Universal Robots PolyScope program: 1ac.urp

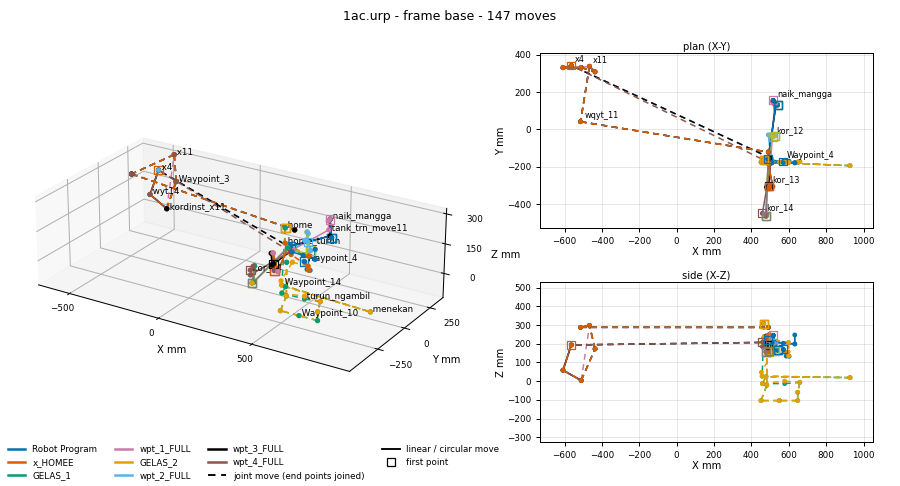
[picture p0: tool path of 1ac.urp in frame base, 147 of 147 moves have a stored position in this frame; points joined in program order, loops and branches not executed]
Program 1ac (createdIn=3.4.3.361 lastSavedIn=3.4.3.361 directory=/programs installation=default robotSerialNumber=2017332896)
Calibrated DH parameters: a=[0.000025, -0.243644, -0.213352, 0.00001, -0.000078, 0]; d=[0.152306, -2.943792, 4.680366, -1.624115, 0.085414, 0.082498]; alpha=[1.571129, 0.003245, -0.003887, 1.571551, -1.571075, 0]; deltaTheta=[0.000074, -0.039266, 0.00755, 0.031605, -0.000097, -0.000018]
BeforeStart
  komunikasi := socket_open("192.168.0.120",30002)
  count := 0
Robot Program (runOnlyOnce=false motionType=MoveJ speed=1.047198 acceleration=1.396263 useActiveTCP=false)
  MoveJ speed 60 deg/s, acceleration 80 deg/s^2 (useActiveTCP=false)
    SuppressedNode
      Waypoint x_HOME: TCP in base x=391.792 y=-168.42 z=273.232 mm, rx=2.1755 ry=-0.1538 rz=2.2323 rad; joints [-13.452, -76.313, -113.498, -168.909, -98.804, -86.905] deg; flange x=205.883 y=-152.538 z=268.8 mm, rx=0.1091 ry=1.5439 rz=-0.0229 rad
    URCap RG2 (RG2 - On Robot, On Robot ApS) data=depthCompensate = false
      | width = 0
      | name = RG2(0)
      | force = 40
      | trigIsDefined = 1
  Loop While (checkContinuously=false) expression=komunikasi≟ False
    komunikasi := socket_open("192.168.0.120",30002)
    If digital_in[7]≟ False
      MoveJ speed 60 deg/s, acceleration 80 deg/s^2 (useActiveTCP=false)
        Waypoint Waypoint_4: TCP in base x=570.948 y=-172.227 z=170.703 mm, rx=1.2117 ry=1.0902 rz=1.141 rad; joints [-5.248, -122.842, -90.085, -143.869, -88.947, -540.731] deg; flange x=385.83 y=-150.884 z=160.264 mm, rx=-1.1206 ry=1.2455 rz=-1.3283 rad
        Waypoint Waypoint_5: TCP in base x=571.886 y=-168.478 z=167.165 mm, rx=0.1353 ry=1.5152 rz=-0.0293 rad; joints [-4.915, -123.143, -90.137, -143.887, -89.039, -626.132] deg; flange x=386.547 y=-148.493 z=157.904 mm, rx=2.1391 ry=-0.191 rz=2.2564 rad
        Waypoint Waypoint_7: TCP in base x=585.683 y=-169.223 z=134.026 mm, rx=0.0805 ry=1.5489 rz=0.0242 rad; joints [-8.112, -130.965, -83.945, -143.962, -96.278, -626.137] deg; flange x=399.213 y=-162.362 z=130.346 mm, rx=-2.181 ry=0.1133 rz=-2.2277 rad
        Waypoint Waypoint_15: TCP in base x=601.355 y=-170.35 z=133.169 mm, rx=0.1182 ry=1.5455 rz=-0.0126 rad; joints [-5.838, -133.147, -80.115, -145.564, -91.253, -626.166] deg; flange x=415.411 y=-154.657 z=129.279 mm, rx=2.184 ry=-0.1672 rz=2.2361 rad
        Wait DigitalInput pin=digital_in[7]; digitalValue=0
    Wait Sleep waitTime=0.5
  pose_position := get_actual_tcp_pose()
  joint_positions := get_actual_joint_positions()
  Script: socket_send_string(pose_position)
  Wait Sleep waitTime=0.5
  Script: socket_send_string(joint_positions)
  Wait Sleep waitTime=0.5
  Script: socket_send_string("asking_for_data")
  Wait Sleep waitTime=0.5
  dt_kirim := socket_read_ascii_float(1)
  dt_terima := dt_kirim[1]
  Wait Sleep waitTime=0.5
  komunikasi := False
  Script: socket_close()
  Folder Folder
    '1'
    If komunikasi≟ False
      If dt_terima≟1
        MoveJ speed 60 deg/s, acceleration 80 deg/s^2 (useActiveTCP=false)
          If digital_in[4]≟ False
            Call GELAS_1
            Call wpt_1_FULL
          ElseIf digital_in[4]≟ True
            Call GELAS_2
            Call wpt_1_FULL
        dt_terima := 0
      If dt_terima≟2
        MoveJ speed 60 deg/s, acceleration 80 deg/s^2 (useActiveTCP=false)
          If digital_in[4]≟ False
            Call GELAS_1
            Call wpt_2_FULL
          ElseIf digital_in[4]≟ True
            Call GELAS_2
            Call wpt_2_FULL
          dt_terima := 0
      If dt_terima≟3
        MoveJ speed 60 deg/s, acceleration 80 deg/s^2 (useActiveTCP=false)
          If digital_in[4]≟ False
            Call GELAS_1
            Call wpt_3_FULL
          ElseIf digital_in[4]≟ True
            Call GELAS_2
            Call wpt_3_FULL
          dt_terima := 0
      If dt_terima≟4
        MoveJ speed 60 deg/s, acceleration 80 deg/s^2 (useActiveTCP=false)
          If digital_in[4]≟ False
            Call GELAS_1
            Call wpt_4_FULL
          ElseIf digital_in[4]≟ True
            Call GELAS_2
            Call wpt_4_FULL
          dt_terima := 0
      '50=50'
      If dt_terima≟5
        'mangga'
        MoveJ speed 60 deg/s, acceleration 80 deg/s^2 (useActiveTCP=false)
          If digital_in[4]≟ False
            Call GELAS_1
            Call manga50
            Call melon50
            Call mixer
            Call x_to_pelanggan
          ElseIf digital_in[4]≟ True
            Call GELAS_2
            Call manga50
            Call melon50
            Call mixer
            Call x_to_pelanggan
          dt_terima := 0
      If dt_terima≟6
        MoveJ speed 60 deg/s, acceleration 80 deg/s^2 (useActiveTCP=false)
          If digital_in[4]≟ False
            Call GELAS_1
            Call manga50
            Call melon50
            Call mixer
            Call x_to_pelanggan
          ElseIf digital_in[4]≟ True
            Call GELAS_2
            Call manga50
            Call melon50
            Call mixer
            Call x_to_pelanggan
          dt_terima := 0
      If dt_terima≟7
        MoveJ speed 60 deg/s, acceleration 80 deg/s^2 (useActiveTCP=false)
          If digital_in[4]≟ False
            Call GELAS_1
            Call manga50
            Call cc_pandan50
            Call mixer
            Call x_to_pelanggan
          ElseIf digital_in[4]≟ True
            Call GELAS_2
            Call manga50
            Call cc_pandan50
            Call mixer
            Call x_to_pelanggan
          dt_terima := 0
      If dt_terima≟8
        MoveJ speed 60 deg/s, acceleration 80 deg/s^2 (useActiveTCP=false)
          If digital_in[4]≟ False
            Call GELAS_1
            Call melon50
            Call jeruk50
            Call mixer
            Call x_to_pelanggan
          ElseIf digital_in[4]≟ True
            Call GELAS_2
            Call melon50
            Call jeruk50
            Call mixer
            Call x_to_pelanggan
          dt_terima := 0
      If dt_terima≟9
        MoveJ speed 60 deg/s, acceleration 80 deg/s^2 (useActiveTCP=false)
          If digital_in[4]≟ False
            Call GELAS_1
            Call melon50
            Call cc_pandan50
            Call mixer
            Call x_to_pelanggan
          ElseIf digital_in[4]≟ True
            Call GELAS_2
            Call melon50
            Call cc_pandan50
            Call mixer
            Call x_to_pelanggan
          count := 0
      If dt_terima≟10
        MoveJ speed 60 deg/s, acceleration 80 deg/s^2 (useActiveTCP=false)
          If digital_in[4]≟ False
            Call GELAS_1
            Call melon50
            Call manga50
            Call mixer
            Call x_to_pelanggan
          ElseIf digital_in[4]≟ True
            Call GELAS_2
            Call melon50
            Call manga50
            Call mixer
            Call x_to_pelanggan
          count := 0
      If dt_terima≟11
        MoveJ speed 60 deg/s, acceleration 80 deg/s^2 (useActiveTCP=false)
          If digital_in[4]≟ False
            Call GELAS_1
            Call jeruk50
            Call manga50
            Call mixer
            Call x_to_pelanggan
          ElseIf digital_in[4]≟ True
            Call GELAS_2
            Call jeruk50
            Call manga50
            Call mixer
            Call x_to_pelanggan
          count := 0
      If dt_terima≟12
        MoveJ speed 60 deg/s, acceleration 80 deg/s^2 (useActiveTCP=false)
          If digital_in[4]≟ False
            Call GELAS_1
            Call jeruk50
            Call melon50
            Call mixer
            Call x_to_pelanggan
          ElseIf digital_in[4]≟ True
            Call GELAS_2
            Call jeruk50
            Call melon50
            Call mixer
            Call x_to_pelanggan
          count := 0
      If dt_terima≟13
        MoveJ speed 60 deg/s, acceleration 80 deg/s^2 (useActiveTCP=false)
          If digital_in[4]≟ False
            Call GELAS_1
            Call jeruk50
            Call cc_pandan50
            Call mixer
            Call x_to_pelanggan
          ElseIf digital_in[4]≟ True
            Call GELAS_2
            Call jeruk50
            Call cc_pandan50
            Call mixer
            Call x_to_pelanggan
          count := 0
      If dt_terima≟14
        MoveJ speed 60 deg/s, acceleration 80 deg/s^2 (useActiveTCP=false)
          If digital_in[4]≟ False
            Call GELAS_1
            Call cc_pandan50
            Call manga50
            Call mixer
            Call x_to_pelanggan
          ElseIf digital_in[4]≟ True
            Call GELAS_2
            Call cc_pandan50
            Call manga50
            Call mixer
            Call x_to_pelanggan
          count := 0
      If dt_terima≟15
        MoveJ speed 60 deg/s, acceleration 80 deg/s^2 (useActiveTCP=false)
          If digital_in[4]≟ False
            Call GELAS_1
            Call cc_pandan50
            Call melon50
            Call mixer
            Call x_to_pelanggan
          ElseIf digital_in[4]≟ True
            Call GELAS_2
            Call cc_pandan50
            Call melon50
            Call mixer
            Call x_to_pelanggan
          count := 0
      If dt_terima≟16
        MoveJ speed 60 deg/s, acceleration 80 deg/s^2 (useActiveTCP=false)
          If digital_in[4]≟ False
            Call GELAS_1
            Call cc_pandan50
            Call jeruk50
            Call mixer
            Call x_to_pelanggan
          ElseIf digital_in[4]≟ True
            Call GELAS_2
            Call cc_pandan50
            Call jeruk50
            Call mixer
            Call x_to_pelanggan
          count := 0
      '75:25'
      If dt_terima≟17
        MoveJ speed 60 deg/s, acceleration 80 deg/s^2 (useActiveTCP=false)
          If digital_in[4]≟ False
            Call GELAS_1
            Call cc_pandan75
            Call melon25
            Call mixer
            Call x_to_pelanggan
          ElseIf digital_in[4]≟ True
            Call GELAS_2
            Call manga75
            Call melon25
            Call mixer
            Call x_to_pelanggan
          count := 0
      If dt_terima≟18
        MoveJ speed 60 deg/s, acceleration 80 deg/s^2 (useActiveTCP=false)
          If digital_in[4]≟ False
            Call GELAS_1
            Call manga75
            Call jeruk25
            Call mixer
            Call x_to_pelanggan
          ElseIf digital_in[4]≟ True
            Call GELAS_2
            Call manga75
            Call jeruk25
            Call mixer
            Call x_to_pelanggan
          count := 0
      If dt_terima≟19
        MoveJ speed 60 deg/s, acceleration 80 deg/s^2 (useActiveTCP=false)
          If digital_in[4]≟ False
            Call GELAS_1
            Call manga75
            Call cc_pandan25
            Call mixer
            Call x_to_pelanggan
          ElseIf digital_in[4]≟ True
            Call GELAS_2
            Call manga75
            Call cc_pandan25
            Call mixer
            Call x_to_pelanggan
          count := 0
      If dt_terima≟20
        MoveJ speed 60 deg/s, acceleration 80 deg/s^2 (useActiveTCP=false)
          If digital_in[4]≟ False
            Call GELAS_1
            Call melon75
            Call manga25
            Call mixer
            Call x_to_pelanggan
          ElseIf digital_in[4]≟ True
            Call GELAS_2
            Call melon75
            Call manga25
            Call mixer
            Call x_to_pelanggan
          count := 0
      If dt_terima≟21
        MoveJ speed 60 deg/s, acceleration 80 deg/s^2 (useActiveTCP=false)
          If digital_in[4]≟ False
            Call GELAS_1
            Call melon75
            Call jeruk25
            Call mixer
            Call x_to_pelanggan
          ElseIf digital_in[4]≟ True
            Call GELAS_2
            Call melon75
            Call jeruk25
            Call mixer
            Call x_to_pelanggan
          count := 0
      If dt_terima≟22
        MoveJ speed 60 deg/s, acceleration 80 deg/s^2 (useActiveTCP=false)
          If digital_in[4]≟ False
            Call GELAS_1
            Call manga75
            Call cc_pandan25
            Call mixer
            Call x_to_pelanggan
          ElseIf digital_in[4]≟ True
            Call GELAS_2
            Call melon75
            Call cc_pandan25
            Call mixer
            Call x_to_pelanggan
          count := 0
      If dt_terima≟23
        MoveJ speed 60 deg/s, acceleration 80 deg/s^2 (useActiveTCP=false)
          If digital_in[4]≟ False
            Call GELAS_1
            Call jeruk75
            Call manga25
            Call mixer
            Call x_to_pelanggan
          ElseIf digital_in[4]≟ True
            Call GELAS_2
            Call manga75
            Call melon25
            Call mixer
            Call x_to_pelanggan
          count := 0
      If dt_terima≟24
        MoveJ speed 60 deg/s, acceleration 80 deg/s^2 (useActiveTCP=false)
          If digital_in[4]≟ False
            Call GELAS_1
            Call jeruk75
            Call melon25
            Call mixer
            Call x_to_pelanggan
          ElseIf digital_in[4]≟ True
            Call GELAS_2
            Call jeruk75
            Call melon25
            Call mixer
            Call x_to_pelanggan
          count := 0
      If dt_terima≟25
        MoveJ speed 60 deg/s, acceleration 80 deg/s^2 (useActiveTCP=false)
          If digital_in[4]≟ False
            Call GELAS_1
            Call jeruk75
            Call cc_pandan25
            Call mixer
            Call x_to_pelanggan
          ElseIf digital_in[4]≟ True
            Call GELAS_2
            Call jeruk75
            Call cc_pandan25
            Call mixer
            Call x_to_pelanggan
          count := 0
      If dt_terima≟26
        MoveJ speed 60 deg/s, acceleration 80 deg/s^2 (useActiveTCP=false)
          If digital_in[4]≟ False
            Call GELAS_1
            Call cc_pandan75
            Call manga25
            Call mixer
            Call x_to_pelanggan
          ElseIf digital_in[4]≟ True
            Call GELAS_2
            Call cc_pandan75
            Call manga25
            Call mixer
            Call x_to_pelanggan
          count := 0
      If dt_terima≟27
        MoveJ speed 60 deg/s, acceleration 80 deg/s^2 (useActiveTCP=false)
          If digital_in[4]≟ False
            Call GELAS_1
            Call cc_pandan75
            Call melon25
            Call mixer
            Call x_to_pelanggan
          ElseIf digital_in[4]≟ True
            Call GELAS_2
            Call cc_pandan75
            Call melon25
            Call mixer
            Call x_to_pelanggan
          count := 0
      If dt_terima≟28
        MoveJ speed 60 deg/s, acceleration 80 deg/s^2 (useActiveTCP=false)
          If digital_in[4]≟ False
            Call GELAS_1
            Call cc_pandan75
            Call jeruk25
            Call mixer
            Call x_to_pelanggan
          ElseIf digital_in[4]≟ True
            Call GELAS_2
            Call cc_pandan75
            Call jeruk25
            Call mixer
            Call x_to_pelanggan
          count := 0
SubProgram x_HOMEE (keepSynchronizedWithDisk=false trackProgramExecution=false)
  MoveJ speed 60 deg/s, acceleration 80 deg/s^2 (useActiveTCP=false)
    URCap RG2 (RG2 - On Robot, On Robot ApS) data=depthCompensate = false
      | width = 1
      | name = RG2(1)
      | force = 40
    Waypoint home: TCP in base x=465.781 y=-163.2 z=307.982 mm, rx=2.2131 ry=-0.1438 rz=2.1498 rad; joints [-6.335, -90.349, -88.069, -183.337, -90.61, -448.752] deg; flange x=280.211 y=-144.033 z=313.667 mm, rx=0.1039 ry=1.5981 rz=-0.059 rad
    Waypoint home_turun: TCP in base x=465.77 y=-163.179 z=232.407 mm, rx=2.213 ry=-0.1437 rz=2.1498 rad; joints [-6.338, -93.095, -105.878, -162.781, -90.691, -448.731] deg; flange x=280.211 y=-144.033 z=238.067 mm, rx=0.1039 ry=1.5981 rz=-0.059 rad
    Waypoint atassss_x: TCP in base x=598.112 y=-177.855 z=206.083 mm, rx=2.2119 ry=-0.1427 rz=2.1519 rad; joints [-6.364, -125.294, -68.76, -167.607, -90.711, -448.64] deg; flange x=412.5 y=-158.899 z=211.472 mm, rx=0.1031 ry=1.5965 rz=-0.0584 rad
    URCap RG2 (RG2 - On Robot, On Robot ApS) data=depthCompensate = false
      | width = 1
      | name = RG2(1)
      | force = 40
      | trigIsDefined = 1
    Waypoint Waypoint_11: TCP in base x=598.658 y=-176.907 z=135.661 mm, rx=2.1942 ry=-0.0737 rz=2.2293 rad; joints [-8.81, -133.678, -77.817, -147.642, -96.613, -448.603] deg; flange x=412.203 y=-169.004 z=132.828 mm, rx=0.0522 ry=1.5546 rz=-0.0142 rad
    Waypoint Waypoint_12: TCP in base x=594.94 y=-176.974 z=154.637 mm, rx=2.1941 ry=-0.0738 rz=2.2293 rad; joints [-8.906, -130.676, -77.596, -150.867, -96.705, -448.616] deg; flange x=408.489 y=-169.004 z=151.793 mm, rx=0.0522 ry=1.5546 rz=-0.0142 rad
    Waypoint Waypoint_2: TCP in base x=505.661 y=-176.925 z=191.063 mm, rx=2.1942 ry=-0.0738 rz=2.2294 rad; joints [-11.93, -109.606, -101.219, -148.324, -99.775, -448.622] deg; flange x=319.191 y=-169.004 z=188.193 mm, rx=0.0522 ry=1.5546 rz=-0.0142 rad
    Wait Sleep waitTime=1
SubProgram -> GELAS_1
SubProgram -> GELAS_2
SubProgram -> wpt_1_FULL
SubProgram -> wpt_2_FULL
SubProgram -> wpt_3_FULL
SubProgram -> wpt_4_FULL
SubProgram -> mixer
SubProgram -> x_to_pelanggan
SubProgram -> manga25
SubProgram -> manga50
SubProgram -> manga75
SubProgram -> melon25
SubProgram -> melon50
SubProgram -> melon75
SubProgram -> jeruk25
SubProgram -> jeruk50
SubProgram -> jeruk75
SubProgram -> cc_pandan25
SubProgram -> cc_pandan50
SubProgram -> cc_pandan75
SubProgram GELAS_1 (keepSynchronizedWithDisk=false trackProgramExecution=false)
  Folder ada gelas
    Set DigitalOutput pin=digital_out[5]; digitalValue=1
    Wait DigitalInput pin=digital_in[4]; digitalValue=1
    Set DigitalOutput pin=digital_out[5]; digitalValue=0
    MoveJ speed 60 deg/s, acceleration 80 deg/s^2 (useActiveTCP=false)
      Waypoint home: TCP in base x=465.781 y=-163.2 z=307.982 mm, rx=2.2131 ry=-0.1438 rz=2.1498 rad; joints [-6.335, -90.349, -88.069, -183.337, -90.61, -448.752] deg; flange x=280.211 y=-144.033 z=313.667 mm, rx=0.1039 ry=1.5981 rz=-0.059 rad
      URCap RG2 (RG2 - On Robot, On Robot ApS) data=depthCompensate = false
        | width = 1
        | name = RG2(1)
        | force = 40
        | trigIsDefined = 1
      Waypoint Waypoint_14: TCP in base x=457.281 y=-175.59 z=26.838 mm, rx=1.3125 ry=1.1415 rz=1.2269 rad; joints [-13.594, -134.915, -121.074, -105.254, -101.04, -535.132] deg; flange x=270.934 y=-166.151 z=30.844 mm, rx=-1.1321 ry=1.3016 rz=-1.1711 rad
      Waypoint menekan: TCP in base x=927.287 y=-194.381 z=18.884 mm, rx=1.3123 ry=1.1416 rz=1.227 rad; joints [-9.415, -143.423, -93.965, -123.848, -96.813, -535.091] deg; flange x=368.179 y=-166.241 z=30.674 mm, rx=-1.1321 ry=1.3016 rz=-1.1712 rad
      Waypoint Waypoint_1: TCP in base x=477.628 y=-175.591 z=23.718 mm, rx=1.3124 ry=1.1415 rz=1.2269 rad; joints [-12.45, -136.993, -115.823, -108.423, -99.888, -535.116] deg; flange x=291.266 y=-166.155 z=27.651 mm, rx=-1.1321 ry=1.3016 rz=-1.1712 rad
      Waypoint melepas: TCP in base x=458.411 y=-175.554 z=-13.316 mm, rx=1.3123 ry=1.1415 rz=1.227 rad; joints [-13.508, -145.696, -118.051, -97.486, -100.932, -535.079] deg; flange x=272.025 y=-166.155 z=-9.385 mm, rx=-1.1321 ry=1.3016 rz=-1.1712 rad
      Waypoint turun_ngambil: TCP in base x=577.568 y=-175.591 z=-13.173 mm, rx=1.312 ry=1.1412 rz=1.2271 rad; joints [-8.749, -154.075, -84.016, -123.141, -96.118, -535.057] deg; flange x=391.122 y=-166.155 z=-9.385 mm, rx=-1.1321 ry=1.3016 rz=-1.1712 rad
      URCap RG2 (RG2 - On Robot, On Robot ApS) data=depthCompensate = false
        | width = 80
        | name = RG2(80)
        | force = 40
        | trigIsDefined = 1
      Waypoint ngambil_gls: TCP in base x=658.794 y=-172.982 z=-6.633 mm, rx=1.2113 ry=1.1561 rz=1.1802 rad; joints [-6.678, -167.29, -51.511, -139.786, -93.955, -540.177] deg; flange x=472.478 y=-163.54 z=-11.189 mm, rx=-1.17 ry=1.2257 rz=-1.2612 rad
      URCap RG2 (RG2 - On Robot, On Robot ApS) data=depthCompensate = false
        | width = 65
        | name = RG2(65)
        | force = 40
        | trigIsDefined = 1
      Waypoint pos_tengah: TCP in base x=647.404 y=-175.552 z=-59.605 mm, rx=1.3122 ry=1.1415 rz=1.227 rad; joints [-7.251, -174.072, -49.105, -138.054, -94.522, -535.053] deg; flange x=461.01 y=-166.155 z=-55.726 mm, rx=-1.1321 ry=1.3016 rz=-1.1712 rad
      Waypoint Waypoint_9: TCP in base x=647.35 y=-175.593 z=-103.933 mm, rx=1.3125 ry=1.1416 rz=1.2268 rad; joints [-7.266, -184.318, -39.11, -137.803, -94.505, -535.052] deg; flange x=461.01 y=-166.155 z=-99.95 mm, rx=-1.1321 ry=1.3016 rz=-1.1712 rad
      Waypoint Waypoint_10: TCP in base x=549.634 y=-175.665 z=-103.877 mm, rx=1.3125 ry=1.1413 rz=1.2268 rad; joints [-9.537, -171.048, -81.148, -109.03, -96.876, -535.008] deg; flange x=363.283 y=-166.155 z=-99.95 mm, rx=-1.1321 ry=1.3016 rz=-1.1712 rad
      Waypoint Waypoint_13: TCP in base x=451.14 y=-175.572 z=-103.927 mm, rx=1.3124 ry=1.1415 rz=1.2269 rad; joints [-13.924, -168.898, -106.738, -85.583, -101.277, -535.013] deg; flange x=264.785 y=-166.155 z=-99.95 mm, rx=-1.1321 ry=1.3016 rz=-1.1712 rad
      Waypoint posisi_awal: TCP in base x=482.025 y=-175.493 z=-22.147 mm, rx=1.3123 ry=1.1417 rz=1.227 rad; joints [-12.21, -148.685, -111.388, -101.158, -99.624, -535.06] deg; flange x=295.641 y=-166.159 z=-18.168 mm, rx=-1.1321 ry=1.3016 rz=-1.1712 rad
      Waypoint Waypoint_6: TCP in base x=481.976 y=-175.586 z=146.433 mm, rx=1.2721 ry=1.093 rz=1.266 rad; joints [-12.268, -112.792, -114.18, -130.689, -99.712, -533.952] deg; flange x=295.752 y=-166.196 z=138.888 mm, rx=-1.0808 ry=1.2578 rz=-1.1901 rad
      Wait Sleep waitTime=1
      count := 0
SubProgram wpt_1_FULL (keepSynchronizedWithDisk=false trackProgramExecution=false)
  MoveL speed 900 mm/s, acceleration 2000 mm/s^2 (useActiveTCP=false) feature=Base
    Waypoint naik_mangga: TCP in base x=516.104 y=155.592 z=244.691 mm, rx=1.2197 ry=1.1492 rz=1.1606 rad; joints [57.005, -107.301, -89.016, -161.054, -29.34, -542.902] deg; flange x=329.909 y=168.377 z=241.061 mm, rx=-1.1689 ry=1.2405 rz=-1.2756 rad
    Waypoint naik_mangga_1: TCP in base x=511.576 y=146.98 z=239.351 mm, rx=1.2548 ry=1.1415 rz=1.2674 rad; joints [55.212, -103.658, -95.728, -157.804, -34.165, -537.934] deg; flange x=325.018 y=149.927 z=234.732 mm, rx=-1.1259 ry=1.2376 rz=-1.1738 rad
    Wait Sleep waitTime=3
    Script: stopl(1)
    Set DigitalOutput pin=digital_out[1]; digitalValue=1
    Wait Sleep waitTime=12
    Set DigitalOutput pin=digital_out[1]; digitalValue=0
    Wait Sleep waitTime=3
    Waypoint tank_trn_move11: TCP in base x=523.005 y=133.061 z=201.593 mm, rx=1.2549 ry=1.1076 rz=1.2428 rad; joints [52.625, -109.232, -100.479, -146.181, -34.757, -539.311] deg; flange x=336.748 y=142.707 z=194.407 mm, rx=-1.1026 ry=1.2492 rz=-1.2115 rad
    Waypoint to_pelangn11: TCP in base x=503.907 y=-154.27 z=207.72 mm, rx=1.2089 ry=1.268 rz=1.203 rad; joints [-11.453, -106.609, -96.119, -159.525, -103.535, -541.638] deg; flange x=317.5 y=-160.213 z=214.737 mm, rx=-1.2637 ry=1.2044 rz=-1.1796 rad
    MoveJ speed 60 deg/s, acceleration 80 deg/s^2 (useActiveTCP=false)
      Waypoint x4: TCP in base x=-563.423 y=342.6 z=193.594 mm, rx=1.214 ry=-1.2627 rz=-1.2329 rad; joints [-213.522, -154.33, -17.776, -189.997, -120.91, -541.566] deg; flange x=-377.075 y=334.014 z=199.223 mm, rx=-1.2484 ry=-1.2004 rz=1.1563 rad
    Waypoint wyt14: TCP in base x=-608.264 y=330.914 z=58.539 mm, rx=1.2121 ry=-1.2682 rz=-1.2314 rad; joints [-209.106, -174.035, -12.62, -175.501, -116.328, -541.259] deg; flange x=-421.955 y=321.813 z=64.701 mm, rx=-1.2538 ry=-1.1985 rz=1.1553 rad
    URCap RG2 (RG2 - On Robot, On Robot ApS) data=depthCompensate = false
      | width = 100
      | name = RG2(100)
      | force = 40
      | trigIsDefined = 1
    Waypoint kordinst_x11: TCP in base x=-510.718 y=331.9 z=3.59 mm, rx=1.2144 ry=-1.2627 rz=-1.2333 rad; joints [-216.478, -159.294, -62.16, -140.686, -124.021, -541.651] deg; flange x=-324.395 y=323.263 z=9.31 mm, rx=-1.2481 ry=-1.2005 rz=1.1559 rad
    MoveJ speed 60 deg/s, acceleration 80 deg/s^2 (useActiveTCP=false)
      Waypoint x11: TCP in base x=-466.424 y=338.501 z=297.896 mm, rx=0.941 ry=-1.628 rz=-1.5836 rad; joints [-198.809, -108.736, -68.355, -185.153, -77.9, -540.869] deg; flange x=-306.703 y=242.215 z=305.123 mm, rx=-1.4425 ry=-0.8338 rz=0.7745 rad
      Waypoint wqyt_11: TCP in base x=-514.336 y=41.381 z=287.863 mm, rx=1.2533 ry=-1.226 rz=-1.2035 rad; joints [-162.747, -92.93, -90.241, -179.052, -73.069, -540.731] deg; flange x=-327.839 y=41.8 z=295.044 mm, rx=-1.2215 ry=-1.2484 rz=1.1782 rad
      Waypoint Way11: TCP in base x=490.038 y=-121.313 z=287.624 mm, rx=1.2437 ry=1.2229 rz=1.1657 rad; joints [-0.404, -92.952, -90.238, -179.048, -89.126, -540.731] deg; flange x=303.606 y=-116.547 z=294.912 mm, rx=-1.2319 ry=1.2529 rz=-1.2153 rad
SubProgram GELAS_2 (keepSynchronizedWithDisk=false trackProgramExecution=false)
  Folder ga ada gelas
    MoveJ speed 60 deg/s, acceleration 80 deg/s^2 (useActiveTCP=false)
      URCap RG2 (RG2 - On Robot, On Robot ApS) data=depthCompensate = false
        | width = 1
        | name = RG2(1)
        | force = 40
      Waypoint home: TCP in base x=465.781 y=-163.2 z=307.982 mm, rx=2.2131 ry=-0.1438 rz=2.1498 rad; joints [-6.335, -90.349, -88.069, -183.337, -90.61, -448.752] deg; flange x=280.211 y=-144.033 z=313.667 mm, rx=0.1039 ry=1.5981 rz=-0.059 rad
      Waypoint home_turun: TCP in base x=465.77 y=-163.179 z=232.407 mm, rx=2.213 ry=-0.1437 rz=2.1498 rad; joints [-6.338, -93.095, -105.878, -162.781, -90.691, -448.731] deg; flange x=280.211 y=-144.033 z=238.067 mm, rx=0.1039 ry=1.5981 rz=-0.059 rad
      Waypoint atassss_x: TCP in base x=598.112 y=-177.855 z=206.083 mm, rx=2.2119 ry=-0.1427 rz=2.1519 rad; joints [-6.364, -125.294, -68.76, -167.607, -90.711, -448.64] deg; flange x=412.5 y=-158.899 z=211.472 mm, rx=0.1031 ry=1.5965 rz=-0.0584 rad
      URCap RG2 (RG2 - On Robot, On Robot ApS) data=depthCompensate = false
        | width = 1
        | name = RG2(1)
        | force = 40
        | trigIsDefined = 1
      Waypoint Waypoint_11: TCP in base x=598.658 y=-176.907 z=135.661 mm, rx=2.1942 ry=-0.0737 rz=2.2293 rad; joints [-8.81, -133.678, -77.817, -147.642, -96.613, -448.603] deg; flange x=412.203 y=-169.004 z=132.828 mm, rx=0.0522 ry=1.5546 rz=-0.0142 rad
      Waypoint Waypoint_12: TCP in base x=594.94 y=-176.974 z=154.637 mm, rx=2.1941 ry=-0.0738 rz=2.2293 rad; joints [-8.906, -130.676, -77.596, -150.867, -96.705, -448.616] deg; flange x=408.489 y=-169.004 z=151.793 mm, rx=0.0522 ry=1.5546 rz=-0.0142 rad
      Waypoint home_x_ats: TCP in base x=512.866 y=-176.962 z=154.673 mm, rx=2.1941 ry=-0.0738 rz=2.2293 rad; joints [-11.608, -115.926, -103.461, -139.754, -99.47, -448.588] deg; flange x=326.409 y=-169.004 z=151.793 mm, rx=0.0522 ry=1.5546 rz=-0.0142 rad
      Waypoint x_blkng: TCP in base x=453.207 y=-175.701 z=47.278 mm, rx=-2.2504 ry=0.0584 rz=-2.1844 rad; joints [-15.793, -129.166, -120.891, -111.742, -104.844, -448.786] deg; flange x=266.71 y=-171.492 z=52.889 mm, rx=0.0415 ry=1.6004 rz=0.0054 rad
      Waypoint Waypoint_14: TCP in base x=457.281 y=-175.59 z=26.838 mm, rx=1.3125 ry=1.1415 rz=1.2269 rad; joints [-13.594, -134.915, -121.074, -105.254, -101.04, -535.132] deg; flange x=270.934 y=-166.151 z=30.844 mm, rx=-1.1321 ry=1.3016 rz=-1.1711 rad
      Waypoint menekan: TCP in base x=927.287 y=-194.381 z=18.884 mm, rx=1.3123 ry=1.1416 rz=1.227 rad; joints [-9.415, -143.423, -93.965, -123.848, -96.813, -535.091] deg; flange x=368.179 y=-166.241 z=30.674 mm, rx=-1.1321 ry=1.3016 rz=-1.1712 rad
      Waypoint ke_blkg_ambl: TCP in base x=477.628 y=-175.591 z=23.718 mm, rx=1.3124 ry=1.1415 rz=1.2269 rad; joints [-12.45, -136.993, -115.823, -108.423, -99.888, -535.116] deg; flange x=291.266 y=-166.155 z=27.651 mm, rx=-1.1321 ry=1.3016 rz=-1.1712 rad
      Waypoint turun_ambl: TCP in base x=458.411 y=-175.554 z=-13.316 mm, rx=1.3123 ry=1.1415 rz=1.227 rad; joints [-13.508, -145.696, -118.051, -97.486, -100.932, -535.079] deg; flange x=272.025 y=-166.155 z=-9.385 mm, rx=-1.1321 ry=1.3016 rz=-1.1712 rad
      Waypoint mju_ngambil: TCP in base x=577.445 y=-175.572 z=0.52 mm, rx=1.2509 ry=1.1298 rz=1.2196 rad; joints [-8.706, -153.211, -85.604, -119.839, -96.03, -536.975] deg; flange x=391.139 y=-166.002 z=-3.801 mm, rx=-1.1299 ry=1.2509 rz=-1.2209 rad
      URCap RG2 (RG2 - On Robot, On Robot ApS) data=depthCompensate = false
        | width = 80
        | name = RG2(80)
        | force = 40
        | trigIsDefined = 1
      Waypoint ngambil_gls: TCP in base x=658.794 y=-172.982 z=-6.633 mm, rx=1.2113 ry=1.1561 rz=1.1802 rad; joints [-6.678, -167.29, -51.511, -139.786, -93.955, -540.177] deg; flange x=472.478 y=-163.54 z=-11.189 mm, rx=-1.17 ry=1.2257 rz=-1.2612 rad
      URCap RG2 (RG2 - On Robot, On Robot ApS) data=depthCompensate = false
        | width = 67
        | name = RG2(67)
        | force = 40
        | trigIsDefined = 1
      Waypoint pos_tengah: TCP in base x=647.404 y=-175.552 z=-59.605 mm, rx=1.3122 ry=1.1415 rz=1.227 rad; joints [-7.251, -174.072, -49.105, -138.054, -94.522, -535.053] deg; flange x=461.01 y=-166.155 z=-55.726 mm, rx=-1.1321 ry=1.3016 rz=-1.1712 rad
      Waypoint Waypoint_9: TCP in base x=647.35 y=-175.593 z=-103.933 mm, rx=1.3125 ry=1.1416 rz=1.2268 rad; joints [-7.266, -184.318, -39.11, -137.803, -94.505, -535.052] deg; flange x=461.01 y=-166.155 z=-99.95 mm, rx=-1.1321 ry=1.3016 rz=-1.1712 rad
      Waypoint Waypoint_10: TCP in base x=549.634 y=-175.665 z=-103.877 mm, rx=1.3125 ry=1.1413 rz=1.2268 rad; joints [-9.537, -171.048, -81.148, -109.03, -96.876, -535.008] deg; flange x=363.283 y=-166.155 z=-99.95 mm, rx=-1.1321 ry=1.3016 rz=-1.1712 rad
      Waypoint Waypoint_13: TCP in base x=451.14 y=-175.572 z=-103.927 mm, rx=1.3124 ry=1.1415 rz=1.2269 rad; joints [-13.924, -168.898, -106.738, -85.583, -101.277, -535.013] deg; flange x=264.785 y=-166.155 z=-99.95 mm, rx=-1.1321 ry=1.3016 rz=-1.1712 rad
      Waypoint posisi_awal: TCP in base x=482.025 y=-175.493 z=-22.147 mm, rx=1.3123 ry=1.1417 rz=1.227 rad; joints [-12.21, -148.685, -111.388, -101.158, -99.624, -535.06] deg; flange x=295.641 y=-166.159 z=-18.168 mm, rx=-1.1321 ry=1.3016 rz=-1.1712 rad
      Waypoint Waypoint_6: TCP in base x=481.976 y=-175.586 z=146.433 mm, rx=1.2721 ry=1.093 rz=1.266 rad; joints [-12.268, -112.792, -114.18, -130.689, -99.712, -533.952] deg; flange x=295.752 y=-166.196 z=138.888 mm, rx=-1.0808 ry=1.2578 rz=-1.1901 rad
      Wait Sleep waitTime=1
      count := 0
SubProgram wpt_2_FULL (keepSynchronizedWithDisk=false trackProgramExecution=false)
  MoveL speed 900 mm/s, acceleration 2000 mm/s^2 (useActiveTCP=false) feature=Base
    Waypoint kor_12: TCP in base x=513.949 y=-40.538 z=204.237 mm, rx=1.201 ry=1.2774 rz=1.1888 rad; joints [15.597, -98.195, -107.467, -156.748, -76.433, -541.429] deg; flange x=327.558 y=-46.238 z=212.053 mm, rx=-1.2774 ry=1.2011 rz=-1.1896 rad
    Waypoint x_tank_2: TCP in base x=506.515 y=-27.084 z=238.197 mm, rx=1.2257 ry=1.2456 rz=1.1731 rad; joints [21.9, -92.41, -104.233, -165.747, -68.149, -540.474] deg; flange x=320.039 y=-26.404 z=245.686 mm, rx=-1.2518 ry=1.2319 rz=-1.2067 rad
    Wait Sleep waitTime=3
    Script: stopl(1)
    Set DigitalOutput pin=digital_out[0]; digitalValue=1
    Wait Sleep waitTime=19
    Set DigitalOutput pin=digital_out[0]; digitalValue=0
    Wait Sleep waitTime=3
    Waypoint tank_trn_move12: TCP in base x=489.882 y=-28.909 z=201.051 mm, rx=1.1185 ry=1.3629 rz=1.2947 rad; joints [10.465, -95.261, -113.119, -153.071, -89.304, -541.973] deg; flange x=305.85 y=-59.703 z=205.796 mm, rx=-1.3236 ry=1.0863 rz=-1.0984 rad
    Waypoint to_pelangn11: TCP in base x=503.907 y=-154.27 z=207.72 mm, rx=1.2089 ry=1.268 rz=1.203 rad; joints [-11.453, -106.609, -96.119, -159.525, -103.535, -541.638] deg; flange x=317.5 y=-160.213 z=214.737 mm, rx=-1.2637 ry=1.2044 rz=-1.1796 rad
    MoveJ speed 60 deg/s, acceleration 80 deg/s^2 (useActiveTCP=false)
      Waypoint x4: TCP in base x=-563.423 y=342.6 z=193.594 mm, rx=1.214 ry=-1.2627 rz=-1.2329 rad; joints [-213.522, -154.33, -17.776, -189.997, -120.91, -541.566] deg; flange x=-377.075 y=334.014 z=199.223 mm, rx=-1.2484 ry=-1.2004 rz=1.1563 rad
    Waypoint wyt14: TCP in base x=-608.264 y=330.914 z=58.539 mm, rx=1.2121 ry=-1.2682 rz=-1.2314 rad; joints [-209.106, -174.035, -12.62, -175.501, -116.328, -541.259] deg; flange x=-421.955 y=321.813 z=64.701 mm, rx=-1.2538 ry=-1.1985 rz=1.1553 rad
    URCap RG2 (RG2 - On Robot, On Robot ApS) data=depthCompensate = false
      | width = 100
      | name = RG2(100)
      | force = 40
      | trigIsDefined = 1
    Waypoint kordinst_x11: TCP in base x=-510.718 y=331.9 z=3.59 mm, rx=1.2144 ry=-1.2627 rz=-1.2333 rad; joints [-216.478, -159.294, -62.16, -140.686, -124.021, -541.651] deg; flange x=-324.395 y=323.263 z=9.31 mm, rx=-1.2481 ry=-1.2005 rz=1.1559 rad
    MoveJ speed 60 deg/s, acceleration 80 deg/s^2 (useActiveTCP=false)
      Waypoint Waypoint_3: TCP in base x=-436.551 y=308.632 z=172.752 mm, rx=1.1669 ry=-1.2108 rz=-1.3302 rad; joints [-219.596, -121.693, -91.009, -143.815, -125.043, -540.78] deg; flange x=-250.818 y=293.104 z=163.21 mm, rx=-1.1764 ry=-1.1337 rz=1.1347 rad
    MoveJ speed 60 deg/s, acceleration 80 deg/s^2 (useActiveTCP=false)
      Waypoint x11: TCP in base x=-466.424 y=338.501 z=297.896 mm, rx=0.941 ry=-1.628 rz=-1.5836 rad; joints [-198.809, -108.736, -68.355, -185.153, -77.9, -540.869] deg; flange x=-306.703 y=242.215 z=305.123 mm, rx=-1.4425 ry=-0.8338 rz=0.7745 rad
      Waypoint wqyt_11: TCP in base x=-514.336 y=41.381 z=287.863 mm, rx=1.2533 ry=-1.226 rz=-1.2035 rad; joints [-162.747, -92.93, -90.241, -179.052, -73.069, -540.731] deg; flange x=-327.839 y=41.8 z=295.044 mm, rx=-1.2215 ry=-1.2484 rz=1.1782 rad
      Waypoint Way11: TCP in base x=490.038 y=-121.313 z=287.624 mm, rx=1.2437 ry=1.2229 rz=1.1657 rad; joints [-0.404, -92.952, -90.238, -179.048, -89.126, -540.731] deg; flange x=303.606 y=-116.547 z=294.912 mm, rx=-1.2319 ry=1.2529 rz=-1.2153 rad
SubProgram wpt_3_FULL (keepSynchronizedWithDisk=false trackProgramExecution=false)
  MoveL speed 900 mm/s, acceleration 2000 mm/s^2 (useActiveTCP=false) feature=Base
    Waypoint kor_13: TCP in base x=490.986 y=-305.163 z=191.28 mm, rx=1.4656 ry=0.8097 rz=0.7645 rad; joints [-9.933, -113.55, -90.212, -159.153, -67.751, -539.356] deg; flange x=333.67 y=-205.151 z=200.248 mm, rx=-0.9154 ry=1.6569 rz=-1.5835 rad
    Waypoint tank_13: TCP in base x=479.978 y=-309.09 z=241.358 mm, rx=1.4657 ry=0.8096 rz=0.7642 rad; joints [-11.106, -108.171, -83.718, -171.001, -68.874, -539.453] deg; flange x=322.714 y=-209.009 z=250.36 mm, rx=-0.9154 ry=1.6571 rz=-1.5836 rad
    Wait Sleep waitTime=3
    Script: stopl(1)
    Set DigitalOutput pin=digital_out[3]; digitalValue=1
    Wait Sleep waitTime=15
    Set DigitalOutput pin=digital_out[3]; digitalValue=0
    Wait Sleep waitTime=3
    Waypoint tank_trn_move13: TCP in base x=490.945 y=-318.144 z=189.866 mm, rx=1.4658 ry=0.8098 rz=0.7643 rad; joints [-12.429, -115.261, -88.008, -159.617, -70.237, -539.486] deg; flange x=333.652 y=-218.105 z=198.922 mm, rx=-0.9155 ry=1.657 rz=-1.5834 rad
    Waypoint to_pelangn11: TCP in base x=503.907 y=-154.27 z=207.72 mm, rx=1.2089 ry=1.268 rz=1.203 rad; joints [-11.453, -106.609, -96.119, -159.525, -103.535, -541.638] deg; flange x=317.5 y=-160.213 z=214.737 mm, rx=-1.2637 ry=1.2044 rz=-1.1796 rad
    MoveJ speed 60 deg/s, acceleration 80 deg/s^2 (useActiveTCP=false)
      Waypoint x4: TCP in base x=-563.423 y=342.6 z=193.594 mm, rx=1.214 ry=-1.2627 rz=-1.2329 rad; joints [-213.522, -154.33, -17.776, -189.997, -120.91, -541.566] deg; flange x=-377.075 y=334.014 z=199.223 mm, rx=-1.2484 ry=-1.2004 rz=1.1563 rad
    Waypoint wyt14: TCP in base x=-608.264 y=330.914 z=58.539 mm, rx=1.2121 ry=-1.2682 rz=-1.2314 rad; joints [-209.106, -174.035, -12.62, -175.501, -116.328, -541.259] deg; flange x=-421.955 y=321.813 z=64.701 mm, rx=-1.2538 ry=-1.1985 rz=1.1553 rad
    URCap RG2 (RG2 - On Robot, On Robot ApS) data=depthCompensate = false
      | width = 100
      | name = RG2(100)
      | force = 40
    Waypoint kordinst_x11: TCP in base x=-510.718 y=331.9 z=3.59 mm, rx=1.2144 ry=-1.2627 rz=-1.2333 rad; joints [-216.478, -159.294, -62.16, -140.686, -124.021, -541.651] deg; flange x=-324.395 y=323.263 z=9.31 mm, rx=-1.2481 ry=-1.2005 rz=1.1559 rad
    MoveJ speed 60 deg/s, acceleration 80 deg/s^2 (useActiveTCP=false)
      Waypoint Waypoint_3: TCP in base x=-436.551 y=308.632 z=172.752 mm, rx=1.1669 ry=-1.2108 rz=-1.3302 rad; joints [-219.596, -121.693, -91.009, -143.815, -125.043, -540.78] deg; flange x=-250.818 y=293.104 z=163.21 mm, rx=-1.1764 ry=-1.1337 rz=1.1347 rad
    MoveJ speed 60 deg/s, acceleration 80 deg/s^2 (useActiveTCP=false)
      Waypoint x11: TCP in base x=-466.424 y=338.501 z=297.896 mm, rx=0.941 ry=-1.628 rz=-1.5836 rad; joints [-198.809, -108.736, -68.355, -185.153, -77.9, -540.869] deg; flange x=-306.703 y=242.215 z=305.123 mm, rx=-1.4425 ry=-0.8338 rz=0.7745 rad
      Waypoint wqyt_11: TCP in base x=-514.336 y=41.381 z=287.863 mm, rx=1.2533 ry=-1.226 rz=-1.2035 rad; joints [-162.747, -92.93, -90.241, -179.052, -73.069, -540.731] deg; flange x=-327.839 y=41.8 z=295.044 mm, rx=-1.2215 ry=-1.2484 rz=1.1782 rad
      Waypoint Way11: TCP in base x=490.038 y=-121.313 z=287.624 mm, rx=1.2437 ry=1.2229 rz=1.1657 rad; joints [-0.404, -92.952, -90.238, -179.048, -89.126, -540.731] deg; flange x=303.606 y=-116.547 z=294.912 mm, rx=-1.2319 ry=1.2529 rz=-1.2153 rad
SubProgram wpt_4_FULL (keepSynchronizedWithDisk=false trackProgramExecution=false)
  MoveL speed 900 mm/s, acceleration 2000 mm/s^2 (useActiveTCP=false) feature=Base
    Waypoint kor_14: TCP in base x=458.532 y=-450.396 z=208.889 mm, rx=1.4426 ry=0.6527 rz=0.6321 rad; joints [-28.206, -127.679, -67.731, -163.247, -75.743, -541.839] deg; flange x=321.375 y=-323.909 z=204.754 mm, rx=-0.7732 ry=1.7087 rz=-1.7654 rad
    Waypoint tank_14: TCP in base x=480.269 y=-462.606 z=236.973 mm, rx=1.4426 ry=0.6528 rz=0.6319 rad; joints [-28.296, -133.156, -50.475, -175.044, -75.769, -541.843] deg; flange x=343.07 y=-336.123 z=232.834 mm, rx=-0.7734 ry=1.7091 rz=-1.7654 rad
    Wait Sleep waitTime=3
    Script: stopl(1)
    Set DigitalOutput pin=digital_out[2]; digitalValue=1
    Wait Sleep waitTime=17
    Set DigitalOutput pin=digital_out[2]; digitalValue=0
    Wait Sleep waitTime=3
    Waypoint tank_trn_move14: TCP in base x=458.609 y=-450.34 z=184.808 mm, rx=1.4427 ry=0.6529 rz=0.6323 rad; joints [-28.201, -129.559, -71.229, -157.872, -75.754, -541.827] deg; flange x=321.375 y=-323.909 z=180.746 mm, rx=-0.7732 ry=1.7087 rz=-1.7654 rad
    Waypoint to_pelangn14: TCP in base x=503.915 y=-182.557 z=207.793 mm, rx=1.2087 ry=1.2681 rz=1.2031 rad; joints [-17.23, -110.658, -90.477, -161.195, -109.302, -541.873] deg; flange x=317.535 y=-188.523 z=214.77 mm, rx=-1.2637 ry=1.2042 rz=-1.1797 rad
    MoveJ speed 60 deg/s, acceleration 80 deg/s^2 (useActiveTCP=false)
      Waypoint x4: TCP in base x=-563.423 y=342.6 z=193.594 mm, rx=1.214 ry=-1.2627 rz=-1.2329 rad; joints [-213.522, -154.33, -17.776, -189.997, -120.91, -541.566] deg; flange x=-377.075 y=334.014 z=199.223 mm, rx=-1.2484 ry=-1.2004 rz=1.1563 rad
    Waypoint wyt14: TCP in base x=-608.264 y=330.914 z=58.539 mm, rx=1.2121 ry=-1.2682 rz=-1.2314 rad; joints [-209.106, -174.035, -12.62, -175.501, -116.328, -541.259] deg; flange x=-421.955 y=321.813 z=64.701 mm, rx=-1.2538 ry=-1.1985 rz=1.1553 rad
    URCap RG2 (RG2 - On Robot, On Robot ApS) data=depthCompensate = false
      | width = 100
      | name = RG2(100)
      | force = 40
      | trigIsDefined = 1
    Waypoint kordinst_x11: TCP in base x=-510.718 y=331.9 z=3.59 mm, rx=1.2144 ry=-1.2627 rz=-1.2333 rad; joints [-216.478, -159.294, -62.16, -140.686, -124.021, -541.651] deg; flange x=-324.395 y=323.263 z=9.31 mm, rx=-1.2481 ry=-1.2005 rz=1.1559 rad
    MoveJ speed 60 deg/s, acceleration 80 deg/s^2 (useActiveTCP=false)
      Waypoint Waypoint_3: TCP in base x=-436.551 y=308.632 z=172.752 mm, rx=1.1669 ry=-1.2108 rz=-1.3302 rad; joints [-219.596, -121.693, -91.009, -143.815, -125.043, -540.78] deg; flange x=-250.818 y=293.104 z=163.21 mm, rx=-1.1764 ry=-1.1337 rz=1.1347 rad
    MoveJ speed 60 deg/s, acceleration 80 deg/s^2 (useActiveTCP=false)
      Waypoint x11: TCP in base x=-466.424 y=338.501 z=297.896 mm, rx=0.941 ry=-1.628 rz=-1.5836 rad; joints [-198.809, -108.736, -68.355, -185.153, -77.9, -540.869] deg; flange x=-306.703 y=242.215 z=305.123 mm, rx=-1.4425 ry=-0.8338 rz=0.7745 rad
      Waypoint wqyt_11: TCP in base x=-514.336 y=41.381 z=287.863 mm, rx=1.2533 ry=-1.226 rz=-1.2035 rad; joints [-162.747, -92.93, -90.241, -179.052, -73.069, -540.731] deg; flange x=-327.839 y=41.8 z=295.044 mm, rx=-1.2215 ry=-1.2484 rz=1.1782 rad
      Waypoint Way11: TCP in base x=490.038 y=-121.313 z=287.624 mm, rx=1.2437 ry=1.2229 rz=1.1657 rad; joints [-0.404, -92.952, -90.238, -179.048, -89.126, -540.731] deg; flange x=303.606 y=-116.547 z=294.912 mm, rx=-1.2319 ry=1.2529 rz=-1.2153 rad
SubProgram manga50 (keepSynchronizedWithDisk=false trackProgramExecution=false)
  MoveL speed 250 mm/s, acceleration 1200 mm/s^2 (useActiveTCP=false) feature=Base
    MoveL speed 250 mm/s, acceleration 1200 mm/s^2 (useActiveTCP=false) feature=Base
      Waypoint manga1_bawah: TCP in base x=539.646 y=130.914 z=166.37 mm, rx=1.1871 ry=1.1862 rz=1.2015 rad; joints [48.394, -115.712, -100.803, -141.071, -41.136, -542.646] deg; flange x=353.092 y=133.446 z=161.548 mm, rx=-1.193 ry=1.1941 rz=-1.2411 rad
    Waypoint naik_mangga: TCP in base x=516.104 y=155.592 z=244.691 mm, rx=1.2197 ry=1.1492 rz=1.1606 rad; joints [57.005, -107.301, -89.016, -161.054, -29.34, -542.902] deg; flange x=329.909 y=168.377 z=241.061 mm, rx=-1.1689 ry=1.2405 rz=-1.2756 rad
    Set DigitalOutput pin=digital_out[1]; digitalValue=1
    Wait Sleep waitTime=6
    Set DigitalOutput pin=digital_out[1]; digitalValue=0
    Wait Sleep waitTime=2
    Waypoint turun_x_tank: TCP in base x=531.003 y=132.408 z=172.736 mm, rx=1.1872 ry=1.1861 rz=1.2015 rad; joints [49.959, -113.318, -102.484, -141.691, -39.573, -542.762] deg; flange x=344.436 y=135 z=167.908 mm, rx=-1.193 ry=1.1942 rz=-1.2411 rad
    MoveL speed 250 mm/s, acceleration 1200 mm/s^2 (useActiveTCP=false) feature=Base
      Waypoint x_tank_home: motionParameters(blendRadius=0.05); TCP in base x=488.881 y=-156.805 z=221.027 mm, rx=1.2554 ry=1.2041 rz=1.1476 rad; joints [-7.578, -99.78, -100.909, -161.579, -94.941, -540.928] deg; flange x=302.63 y=-147.349 z=228.234 mm, rx=-1.2197 ry=1.2715 rz=-1.2332 rad
SubProgram melon50 (keepSynchronizedWithDisk=false trackProgramExecution=false)
  MoveL speed 250 mm/s, acceleration 1200 mm/s^2 (useActiveTCP=false) feature=Base
    Waypoint turun_x2: TCP in base x=523.919 y=-35.076 z=160.824 mm, rx=1.2485 ry=1.2153 rz=1.1584 rad; joints [20.424, -105.524, -112.1, -144.725, -67.852, -539.776] deg; flange x=337.524 y=-28.42 z=168.091 mm, rx=-1.227 ry=1.2605 rz=-1.2226 rad
    Waypoint naik_x2: TCP in base x=502.576 y=-30.727 z=246.495 mm, rx=1.2485 ry=1.2153 rz=1.1582 rad; joints [23.574, -90.742, -103.726, -167.89, -64.628, -539.734] deg; flange x=316.192 y=-24.039 z=253.773 mm, rx=-1.2271 ry=1.2605 rz=-1.2227 rad
    Set DigitalOutput pin=digital_out[0]; digitalValue=1
    Wait Sleep waitTime=9.5
    Set DigitalOutput pin=digital_out[0]; digitalValue=0
    Wait Sleep waitTime=2
    Waypoint turun_x2_tank: TCP in base x=511.293 y=-38.271 z=141.227 mm, rx=1.2483 ry=1.2153 rz=1.1585 rad; joints [20.786, -106.203, -118.142, -138.004, -67.516, -539.739] deg; flange x=324.897 y=-31.646 z=148.465 mm, rx=-1.2268 ry=1.2603 rz=-1.2225 rad
    MoveJ speed 60 deg/s, acceleration 80 deg/s^2 (useActiveTCP=false)
      Waypoint x2_tank_home: TCP in base x=488.881 y=-181.074 z=220.885 mm, rx=1.2486 ry=1.2154 rz=1.1583 rad; joints [-14.048, -103.798, -95.907, -162.637, -102.237, -541.211] deg; flange x=302.517 y=-174.422 z=228.204 mm, rx=-1.227 ry=1.2605 rz=-1.2226 rad
SubProgram mixer (keepSynchronizedWithDisk=false trackProgramExecution=false)
  MoveL speed 250 mm/s, acceleration 1200 mm/s^2 (useActiveTCP=false) feature=Base
    Waypoint x_tank_home: TCP in base x=488.881 y=-156.805 z=221.027 mm, rx=1.2554 ry=1.2041 rz=1.1476 rad; joints [-7.578, -99.78, -100.909, -161.579, -94.941, -540.928] deg; flange x=302.63 y=-147.349 z=228.234 mm, rx=-1.2197 ry=1.2715 rz=-1.2332 rad
    Waypoint Waypoint_18: TCP in base x=569.834 y=-179.096 z=202.81 mm, rx=1.2483 ry=1.215 rz=1.1583 rad; joints [-10.289, -121.136, -75.827, -165.337, -98.443, -541.011] deg; flange x=383.389 y=-172.392 z=209.886 mm, rx=-1.2271 ry=1.2607 rz=-1.2226 rad
    Waypoint Waypoint_19: TCP in base x=631.659 y=-179.11 z=198.561 mm, rx=1.2487 ry=1.2152 rz=1.1582 rad; joints [-8.66, -136.239, -50.831, -175.21, -96.75, -540.914] deg; flange x=445.294 y=-172.375 z=205.884 mm, rx=-1.227 ry=1.2606 rz=-1.2226 rad
    Waypoint Waypoint_20: TCP in base x=631.66 y=-179.046 z=247.147 mm, rx=1.2486 ry=1.2154 rz=1.1582 rad; joints [-8.677, -136.039, -38.139, -188.105, -96.713, -540.914] deg; flange x=445.286 y=-172.392 z=254.415 mm, rx=-1.227 ry=1.2607 rz=-1.2226 rad
    Set DigitalOutput pin=digital_out[4]; digitalValue=1
    Wait Sleep waitTime=5
    Set DigitalOutput pin=digital_out[4]; digitalValue=0
    Waypoint Waypoint_21: TCP in base x=631.672 y=-179.07 z=199.204 mm, rx=1.2485 ry=1.2154 rz=1.1581 rad; joints [-8.66, -136.216, -50.705, -175.357, -96.753, -540.92] deg; flange x=445.298 y=-172.367 z=206.506 mm, rx=-1.2271 ry=1.2605 rz=-1.2227 rad
    Waypoint Waypoint_22: TCP in base x=511.311 y=-179.038 z=206.145 mm, rx=1.2485 ry=1.2154 rz=1.1582 rad; joints [-12.494, -109.067, -93.069, -160.188, -100.685, -541.13] deg; flange x=324.929 y=-172.375 z=213.436 mm, rx=-1.227 ry=1.2606 rz=-1.2226 rad
    Waypoint x_tank_home: TCP in base x=488.881 y=-156.805 z=221.027 mm, rx=1.2554 ry=1.2041 rz=1.1476 rad; joints [-7.578, -99.78, -100.909, -161.579, -94.941, -540.928] deg; flange x=302.63 y=-147.349 z=228.234 mm, rx=-1.2197 ry=1.2715 rz=-1.2332 rad
SubProgram x_to_pelanggan (keepSynchronizedWithDisk=false trackProgramExecution=false)
  MoveJ speed 60 deg/s, acceleration 80 deg/s^2 (useActiveTCP=false)
    Waypoint x4: TCP in base x=-563.423 y=342.6 z=193.594 mm, rx=1.214 ry=-1.2627 rz=-1.2329 rad; joints [-213.522, -154.33, -17.776, -189.997, -120.91, -541.566] deg; flange x=-377.075 y=334.014 z=199.223 mm, rx=-1.2484 ry=-1.2004 rz=1.1563 rad
  MoveJ speed 60 deg/s, acceleration 80 deg/s^2 (useActiveTCP=false)
    Waypoint wyt14: TCP in base x=-608.264 y=330.914 z=58.539 mm, rx=1.2121 ry=-1.2682 rz=-1.2314 rad; joints [-209.106, -174.035, -12.62, -175.501, -116.328, -541.259] deg; flange x=-421.955 y=321.813 z=64.701 mm, rx=-1.2538 ry=-1.1985 rz=1.1553 rad
    URCap RG2 (RG2 - On Robot, On Robot ApS) data=depthCompensate = false
      | width = 100
      | name = RG2(100)
      | force = 40
      | trigIsDefined = 1
    Waypoint kordinst_x11: TCP in base x=-510.718 y=331.9 z=3.59 mm, rx=1.2144 ry=-1.2627 rz=-1.2333 rad; joints [-216.478, -159.294, -62.16, -140.686, -124.021, -541.651] deg; flange x=-324.395 y=323.263 z=9.31 mm, rx=-1.2481 ry=-1.2005 rz=1.1559 rad
    MoveJ speed 60 deg/s, acceleration 80 deg/s^2 (useActiveTCP=false)
      Waypoint Waypoint_3: TCP in base x=-436.551 y=308.632 z=172.752 mm, rx=1.1669 ry=-1.2108 rz=-1.3302 rad; joints [-219.596, -121.693, -91.009, -143.815, -125.043, -540.78] deg; flange x=-250.818 y=293.104 z=163.21 mm, rx=-1.1764 ry=-1.1337 rz=1.1347 rad
    MoveJ speed 60 deg/s, acceleration 80 deg/s^2 (useActiveTCP=false)
      Waypoint x11: TCP in base x=-466.424 y=338.501 z=297.896 mm, rx=0.941 ry=-1.628 rz=-1.5836 rad; joints [-198.809, -108.736, -68.355, -185.153, -77.9, -540.869] deg; flange x=-306.703 y=242.215 z=305.123 mm, rx=-1.4425 ry=-0.8338 rz=0.7745 rad
      Waypoint wqyt_11: TCP in base x=-514.336 y=41.381 z=287.863 mm, rx=1.2533 ry=-1.226 rz=-1.2035 rad; joints [-162.747, -92.93, -90.241, -179.052, -73.069, -540.731] deg; flange x=-327.839 y=41.8 z=295.044 mm, rx=-1.2215 ry=-1.2484 rz=1.1782 rad
      Waypoint Way11: TCP in base x=490.038 y=-121.313 z=287.624 mm, rx=1.2437 ry=1.2229 rz=1.1657 rad; joints [-0.404, -92.952, -90.238, -179.048, -89.126, -540.731] deg; flange x=303.606 y=-116.547 z=294.912 mm, rx=-1.2319 ry=1.2529 rz=-1.2153 rad
SubProgram cc_pandan50 (keepSynchronizedWithDisk=false trackProgramExecution=false)
  MoveL speed 250 mm/s, acceleration 1200 mm/s^2 (useActiveTCP=false) feature=Base
    Waypoint turun_x4: TCP in base x=477.966 y=-466.243 z=156.94 mm, rx=1.4882 ry=0.7462 rz=0.7026 rad; joints [-32.79, -139.243, -56.042, -167.441, -85.85, -540.295] deg; flange x=329.261 y=-353.791 z=165.786 mm, rx=-0.8586 ry=1.7127 rz=-1.6385 rad
    Waypoint naik_x4: TCP in base x=482.264 y=-454.304 z=236.456 mm, rx=1.4042 ry=0.7616 rz=0.7787 rad; joints [-33.695, -133.947, -49.546, -175.016, -90.654, -540.261] deg; flange x=326.118 y=-352.203 z=231.387 mm, rx=-0.8658 ry=1.5964 rz=-1.6409 rad
    Set DigitalOutput pin=digital_out[2]; digitalValue=1
    Wait Sleep waitTime=6.5
    Set DigitalOutput pin=digital_out[2]; digitalValue=0
    Wait Sleep waitTime=2
    Waypoint turun_x4_tank: TCP in base x=478.055 y=-454.296 z=156.757 mm, rx=1.4884 ry=0.7463 rz=0.7024 rad; joints [-31.253, -136.803, -60.661, -165.277, -84.324, -540.226] deg; flange x=329.366 y=-341.82 z=165.7 mm, rx=-0.8587 ry=1.7129 rz=-1.6384 rad
    MoveL speed 250 mm/s, acceleration 1200 mm/s^2 (useActiveTCP=false) feature=Base
      Waypoint x4_tank_home: TCP in base x=488.881 y=-181.074 z=220.885 mm, rx=1.2486 ry=1.2154 rz=1.1583 rad; joints [-14.048, -103.798, -95.907, -162.637, -102.237, -541.211] deg; flange x=302.517 y=-174.422 z=228.204 mm, rx=-1.227 ry=1.2605 rz=-1.2226 rad
SubProgram jeruk50 (keepSynchronizedWithDisk=false trackProgramExecution=false)
  MoveL speed 250 mm/s, acceleration 1200 mm/s^2 (useActiveTCP=false) feature=Base
    Waypoint turun_x3: TCP in base x=495.704 y=-306.283 z=159.319 mm, rx=1.4128 ry=0.9228 rz=0.8745 rad; joints [-17.368, -118.985, -91.708, -151.812, -83.555, -540.246] deg; flange x=325.42 y=-230.264 z=167.468 mm, rx=-1.0113 ry=1.5485 rz=-1.4888 rad
    Waypoint naik_x3: TCP in base x=494.063 y=-315.696 z=248.345 mm, rx=1.4127 ry=0.9226 rz=0.8745 rad; joints [-19.174, -113.016, -75.356, -174.123, -85.284, -540.374] deg; flange x=323.815 y=-239.623 z=256.391 mm, rx=-1.0113 ry=1.5485 rz=-1.4889 rad
    Set DigitalOutput pin=digital_out[3]; digitalValue=1
    Wait Sleep waitTime=8
    Set DigitalOutput pin=digital_out[3]; digitalValue=0
    Wait Sleep waitTime=2
    Waypoint turun_x3_tank: TCP in base x=514.431 y=-306.379 z=159.337 mm, rx=1.4128 ry=0.9227 rz=0.8744 rad; joints [-16.345, -122.244, -86.272, -153.993, -82.521, -540.196] deg; flange x=344.203 y=-230.264 z=167.468 mm, rx=-1.0113 ry=1.5485 rz=-1.4888 rad
    MoveL speed 250 mm/s, acceleration 1200 mm/s^2 (useActiveTCP=false) feature=Base
      Waypoint x3_tank_home: TCP in base x=488.881 y=-181.074 z=220.885 mm, rx=1.2486 ry=1.2154 rz=1.1583 rad; joints [-14.048, -103.798, -95.907, -162.637, -102.237, -541.211] deg; flange x=302.517 y=-174.422 z=228.204 mm, rx=-1.227 ry=1.2605 rz=-1.2226 rad
SubProgram cc_pandan75 (keepSynchronizedWithDisk=false trackProgramExecution=false)
  MoveL speed 250 mm/s, acceleration 1200 mm/s^2 (useActiveTCP=false) feature=Base
    Waypoint turun_x4: TCP in base x=477.966 y=-466.243 z=156.94 mm, rx=1.4882 ry=0.7462 rz=0.7026 rad; joints [-32.79, -139.243, -56.042, -167.441, -85.85, -540.295] deg; flange x=329.261 y=-353.791 z=165.786 mm, rx=-0.8586 ry=1.7127 rz=-1.6385 rad
    Waypoint naik_x4: TCP in base x=482.264 y=-454.304 z=236.456 mm, rx=1.4042 ry=0.7616 rz=0.7787 rad; joints [-33.695, -133.947, -49.546, -175.016, -90.654, -540.261] deg; flange x=326.118 y=-352.203 z=231.387 mm, rx=-0.8658 ry=1.5964 rz=-1.6409 rad
    Set DigitalOutput pin=digital_out[2]; digitalValue=1
    Wait Sleep waitTime=9.75
    Set DigitalOutput pin=digital_out[2]; digitalValue=0
    Wait Sleep waitTime=2
    Waypoint turun_x4_tank: TCP in base x=478.055 y=-454.296 z=156.757 mm, rx=1.4884 ry=0.7463 rz=0.7024 rad; joints [-31.253, -136.803, -60.661, -165.277, -84.324, -540.226] deg; flange x=329.366 y=-341.82 z=165.7 mm, rx=-0.8587 ry=1.7129 rz=-1.6384 rad
    MoveL speed 250 mm/s, acceleration 1200 mm/s^2 (useActiveTCP=false) feature=Base
      Waypoint x4_tank_home: TCP in base x=488.881 y=-181.074 z=220.885 mm, rx=1.2486 ry=1.2154 rz=1.1583 rad; joints [-14.048, -103.798, -95.907, -162.637, -102.237, -541.211] deg; flange x=302.517 y=-174.422 z=228.204 mm, rx=-1.227 ry=1.2605 rz=-1.2226 rad
SubProgram melon25 (keepSynchronizedWithDisk=false trackProgramExecution=false)
  MoveL speed 250 mm/s, acceleration 1200 mm/s^2 (useActiveTCP=false) feature=Base
    Waypoint turun_x2: TCP in base x=523.919 y=-35.076 z=160.824 mm, rx=1.2485 ry=1.2153 rz=1.1584 rad; joints [20.424, -105.524, -112.1, -144.725, -67.852, -539.776] deg; flange x=337.524 y=-28.42 z=168.091 mm, rx=-1.227 ry=1.2605 rz=-1.2226 rad
    Waypoint naik_x2: TCP in base x=502.576 y=-30.727 z=246.495 mm, rx=1.2485 ry=1.2153 rz=1.1582 rad; joints [23.574, -90.742, -103.726, -167.89, -64.628, -539.734] deg; flange x=316.192 y=-24.039 z=253.773 mm, rx=-1.2271 ry=1.2605 rz=-1.2227 rad
    Set DigitalOutput pin=digital_out[0]; digitalValue=1
    Wait Sleep waitTime=4.75
    Set DigitalOutput pin=digital_out[0]; digitalValue=0
    Wait Sleep waitTime=2
    Waypoint turun_x2_tank: TCP in base x=511.293 y=-38.271 z=141.227 mm, rx=1.2483 ry=1.2153 rz=1.1585 rad; joints [20.786, -106.203, -118.142, -138.004, -67.516, -539.739] deg; flange x=324.897 y=-31.646 z=148.465 mm, rx=-1.2268 ry=1.2603 rz=-1.2225 rad
    MoveJ speed 60 deg/s, acceleration 80 deg/s^2 (useActiveTCP=false)
      Waypoint x2_tank_home: TCP in base x=488.881 y=-181.074 z=220.885 mm, rx=1.2486 ry=1.2154 rz=1.1583 rad; joints [-14.048, -103.798, -95.907, -162.637, -102.237, -541.211] deg; flange x=302.517 y=-174.422 z=228.204 mm, rx=-1.227 ry=1.2605 rz=-1.2226 rad
SubProgram manga75 (keepSynchronizedWithDisk=false trackProgramExecution=false)
  MoveL speed 250 mm/s, acceleration 1200 mm/s^2 (useActiveTCP=false) feature=Base
    MoveL speed 250 mm/s, acceleration 1200 mm/s^2 (useActiveTCP=false) feature=Base
      Waypoint manga1_bawah: TCP in base x=539.646 y=130.914 z=166.37 mm, rx=1.1871 ry=1.1862 rz=1.2015 rad; joints [48.394, -115.712, -100.803, -141.071, -41.136, -542.646] deg; flange x=353.092 y=133.446 z=161.548 mm, rx=-1.193 ry=1.1941 rz=-1.2411 rad
    Waypoint naik_mangga: TCP in base x=516.104 y=155.592 z=244.691 mm, rx=1.2197 ry=1.1492 rz=1.1606 rad; joints [57.005, -107.301, -89.016, -161.054, -29.34, -542.902] deg; flange x=329.909 y=168.377 z=241.061 mm, rx=-1.1689 ry=1.2405 rz=-1.2756 rad
    Set DigitalOutput pin=digital_out[1]; digitalValue=1
    Wait Sleep waitTime=9
    Set DigitalOutput pin=digital_out[1]; digitalValue=0
    Wait Sleep waitTime=2
    Waypoint turun_x_tank: TCP in base x=531.003 y=132.408 z=172.736 mm, rx=1.1872 ry=1.1861 rz=1.2015 rad; joints [49.959, -113.318, -102.484, -141.691, -39.573, -542.762] deg; flange x=344.436 y=135 z=167.908 mm, rx=-1.193 ry=1.1942 rz=-1.2411 rad
    MoveL speed 250 mm/s, acceleration 1200 mm/s^2 (useActiveTCP=false) feature=Base
      Waypoint x_tank_home: motionParameters(blendRadius=0.05); TCP in base x=488.881 y=-156.805 z=221.027 mm, rx=1.2554 ry=1.2041 rz=1.1476 rad; joints [-7.578, -99.78, -100.909, -161.579, -94.941, -540.928] deg; flange x=302.63 y=-147.349 z=228.234 mm, rx=-1.2197 ry=1.2715 rz=-1.2332 rad
SubProgram jeruk25 (keepSynchronizedWithDisk=false trackProgramExecution=false)
  MoveL speed 250 mm/s, acceleration 1200 mm/s^2 (useActiveTCP=false) feature=Base
    Waypoint turun_x3: TCP in base x=495.704 y=-306.283 z=159.319 mm, rx=1.4128 ry=0.9228 rz=0.8745 rad; joints [-17.368, -118.985, -91.708, -151.812, -83.555, -540.246] deg; flange x=325.42 y=-230.264 z=167.468 mm, rx=-1.0113 ry=1.5485 rz=-1.4888 rad
    Waypoint naik_x3: TCP in base x=494.063 y=-315.696 z=248.345 mm, rx=1.4127 ry=0.9226 rz=0.8745 rad; joints [-19.174, -113.016, -75.356, -174.123, -85.284, -540.374] deg; flange x=323.815 y=-239.623 z=256.391 mm, rx=-1.0113 ry=1.5485 rz=-1.4889 rad
    Set DigitalOutput pin=digital_out[3]; digitalValue=1
    Wait Sleep waitTime=4
    Set DigitalOutput pin=digital_out[3]; digitalValue=0
    Wait Sleep waitTime=2
    Waypoint turun_x3_tank: TCP in base x=514.431 y=-306.379 z=159.337 mm, rx=1.4128 ry=0.9227 rz=0.8744 rad; joints [-16.345, -122.244, -86.272, -153.993, -82.521, -540.196] deg; flange x=344.203 y=-230.264 z=167.468 mm, rx=-1.0113 ry=1.5485 rz=-1.4888 rad
    MoveL speed 250 mm/s, acceleration 1200 mm/s^2 (useActiveTCP=false) feature=Base
      Waypoint x3_tank_home: TCP in base x=488.881 y=-181.074 z=220.885 mm, rx=1.2486 ry=1.2154 rz=1.1583 rad; joints [-14.048, -103.798, -95.907, -162.637, -102.237, -541.211] deg; flange x=302.517 y=-174.422 z=228.204 mm, rx=-1.227 ry=1.2605 rz=-1.2226 rad
SubProgram cc_pandan25 (keepSynchronizedWithDisk=false trackProgramExecution=false)
  MoveL speed 250 mm/s, acceleration 1200 mm/s^2 (useActiveTCP=false) feature=Base
    Waypoint turun_x4: TCP in base x=477.966 y=-466.243 z=156.94 mm, rx=1.4882 ry=0.7462 rz=0.7026 rad; joints [-32.79, -139.243, -56.042, -167.441, -85.85, -540.295] deg; flange x=329.261 y=-353.791 z=165.786 mm, rx=-0.8586 ry=1.7127 rz=-1.6385 rad
    Waypoint naik_x4: TCP in base x=482.264 y=-454.304 z=236.456 mm, rx=1.4042 ry=0.7616 rz=0.7787 rad; joints [-33.695, -133.947, -49.546, -175.016, -90.654, -540.261] deg; flange x=326.118 y=-352.203 z=231.387 mm, rx=-0.8658 ry=1.5964 rz=-1.6409 rad
    Set DigitalOutput pin=digital_out[2]; digitalValue=1
    Wait Sleep waitTime=3.25
    Set DigitalOutput pin=digital_out[2]; digitalValue=0
    Wait Sleep waitTime=2
    Waypoint turun_x4_tank: TCP in base x=478.055 y=-454.296 z=156.757 mm, rx=1.4884 ry=0.7463 rz=0.7024 rad; joints [-31.253, -136.803, -60.661, -165.277, -84.324, -540.226] deg; flange x=329.366 y=-341.82 z=165.7 mm, rx=-0.8587 ry=1.7129 rz=-1.6384 rad
    MoveL speed 250 mm/s, acceleration 1200 mm/s^2 (useActiveTCP=false) feature=Base
      Waypoint x4_tank_home: TCP in base x=488.881 y=-181.074 z=220.885 mm, rx=1.2486 ry=1.2154 rz=1.1583 rad; joints [-14.048, -103.798, -95.907, -162.637, -102.237, -541.211] deg; flange x=302.517 y=-174.422 z=228.204 mm, rx=-1.227 ry=1.2605 rz=-1.2226 rad
SubProgram melon75 (keepSynchronizedWithDisk=false trackProgramExecution=false)
  MoveL speed 250 mm/s, acceleration 1200 mm/s^2 (useActiveTCP=false) feature=Base
    Waypoint turun_x2: TCP in base x=523.919 y=-35.076 z=160.824 mm, rx=1.2485 ry=1.2153 rz=1.1584 rad; joints [20.424, -105.524, -112.1, -144.725, -67.852, -539.776] deg; flange x=337.524 y=-28.42 z=168.091 mm, rx=-1.227 ry=1.2605 rz=-1.2226 rad
    Waypoint naik_x2: TCP in base x=502.576 y=-30.727 z=246.495 mm, rx=1.2485 ry=1.2153 rz=1.1582 rad; joints [23.574, -90.742, -103.726, -167.89, -64.628, -539.734] deg; flange x=316.192 y=-24.039 z=253.773 mm, rx=-1.2271 ry=1.2605 rz=-1.2227 rad
    Set DigitalOutput pin=digital_out[0]; digitalValue=1
    Wait Sleep waitTime=14.25
    Set DigitalOutput pin=digital_out[0]; digitalValue=0
    Wait Sleep waitTime=2
    Waypoint turun_x2_tank: TCP in base x=511.293 y=-38.271 z=141.227 mm, rx=1.2483 ry=1.2153 rz=1.1585 rad; joints [20.786, -106.203, -118.142, -138.004, -67.516, -539.739] deg; flange x=324.897 y=-31.646 z=148.465 mm, rx=-1.2268 ry=1.2603 rz=-1.2225 rad
    MoveL speed 250 mm/s, acceleration 1200 mm/s^2 (useActiveTCP=false) feature=Base
      Waypoint x2_tank_home: TCP in base x=488.881 y=-181.074 z=220.885 mm, rx=1.2486 ry=1.2154 rz=1.1583 rad; joints [-14.048, -103.798, -95.907, -162.637, -102.237, -541.211] deg; flange x=302.517 y=-174.422 z=228.204 mm, rx=-1.227 ry=1.2605 rz=-1.2226 rad
SubProgram manga25 (keepSynchronizedWithDisk=false trackProgramExecution=false)
  MoveL speed 250 mm/s, acceleration 1200 mm/s^2 (useActiveTCP=false) feature=Base
    MoveL speed 250 mm/s, acceleration 1200 mm/s^2 (useActiveTCP=false) feature=Base
      Waypoint manga1_bawah: TCP in base x=539.646 y=130.914 z=166.37 mm, rx=1.1871 ry=1.1862 rz=1.2015 rad; joints [48.394, -115.712, -100.803, -141.071, -41.136, -542.646] deg; flange x=353.092 y=133.446 z=161.548 mm, rx=-1.193 ry=1.1941 rz=-1.2411 rad
    Waypoint naik_mangga: TCP in base x=516.104 y=155.592 z=244.691 mm, rx=1.2197 ry=1.1492 rz=1.1606 rad; joints [57.005, -107.301, -89.016, -161.054, -29.34, -542.902] deg; flange x=329.909 y=168.377 z=241.061 mm, rx=-1.1689 ry=1.2405 rz=-1.2756 rad
    Set DigitalOutput pin=digital_out[1]; digitalValue=1
    Wait Sleep waitTime=3
    Set DigitalOutput pin=digital_out[1]; digitalValue=0
    Wait Sleep waitTime=2
    Waypoint turun_x_tank: TCP in base x=531.003 y=132.408 z=172.736 mm, rx=1.1872 ry=1.1861 rz=1.2015 rad; joints [49.959, -113.318, -102.484, -141.691, -39.573, -542.762] deg; flange x=344.436 y=135 z=167.908 mm, rx=-1.193 ry=1.1942 rz=-1.2411 rad
    MoveL speed 250 mm/s, acceleration 1200 mm/s^2 (useActiveTCP=false) feature=Base
      Waypoint x_tank_home: motionParameters(blendRadius=0.05); TCP in base x=488.881 y=-156.805 z=221.027 mm, rx=1.2554 ry=1.2041 rz=1.1476 rad; joints [-7.578, -99.78, -100.909, -161.579, -94.941, -540.928] deg; flange x=302.63 y=-147.349 z=228.234 mm, rx=-1.2197 ry=1.2715 rz=-1.2332 rad
SubProgram jeruk75 (keepSynchronizedWithDisk=false trackProgramExecution=false)
  MoveL speed 250 mm/s, acceleration 1200 mm/s^2 (useActiveTCP=false) feature=Base
    Waypoint turun_x3: TCP in base x=495.704 y=-306.283 z=159.319 mm, rx=1.4128 ry=0.9228 rz=0.8745 rad; joints [-17.368, -118.985, -91.708, -151.812, -83.555, -540.246] deg; flange x=325.42 y=-230.264 z=167.468 mm, rx=-1.0113 ry=1.5485 rz=-1.4888 rad
    Waypoint naik_x3: TCP in base x=494.063 y=-315.696 z=248.345 mm, rx=1.4127 ry=0.9226 rz=0.8745 rad; joints [-19.174, -113.016, -75.356, -174.123, -85.284, -540.374] deg; flange x=323.815 y=-239.623 z=256.391 mm, rx=-1.0113 ry=1.5485 rz=-1.4889 rad
    Set DigitalOutput pin=digital_out[3]; digitalValue=1
    Wait Sleep waitTime=12
    Set DigitalOutput pin=digital_out[3]; digitalValue=0
    Wait Sleep waitTime=2
    Waypoint turun_x3_tank: TCP in base x=514.431 y=-306.379 z=159.337 mm, rx=1.4128 ry=0.9227 rz=0.8744 rad; joints [-16.345, -122.244, -86.272, -153.993, -82.521, -540.196] deg; flange x=344.203 y=-230.264 z=167.468 mm, rx=-1.0113 ry=1.5485 rz=-1.4888 rad
    MoveL speed 250 mm/s, acceleration 1200 mm/s^2 (useActiveTCP=false) feature=Base
      Waypoint x3_tank_home: TCP in base x=488.881 y=-181.074 z=220.885 mm, rx=1.2486 ry=1.2154 rz=1.1583 rad; joints [-14.048, -103.798, -95.907, -162.637, -102.237, -541.211] deg; flange x=302.517 y=-174.422 z=228.204 mm, rx=-1.227 ry=1.2605 rz=-1.2226 rad
